{attribute 'linkalways'} 
{attribute 'no_explicit_call' := 'This FB is a CLASS and must be accessed using methods or properties'}
{attribute 'enable_dynamic_creation'}
FUNCTION_BLOCK _ETcVnColorMapSize EXTENDS EnumDatatypeBase
VAR
	localData : ETcVnColorMapSize;
	activeData : REFERENCE TO ETcVnColorMapSize;
	enumBaseDatatype : _UDINT(localData);
END_VAR

METHOD PRIVATE AddLocalEnumeration
VAR_INPUT
	Enumeration : T_MAXSTRING;
	Value : ETcVnColorMapSize;
END_VAR
AddEnumeration(Enumeration, Value);
END_METHOD

PROPERTY PUBLIC Address : PVOID
GET
Address := ADR(activeData);
END_GET
END_PROPERTY

METHOD PUBLIC ClearReference
VAR_INPUT
END_VAR
activeData REF= localData;
SetBaseDatatypeReference();
END_METHOD

METHOD PUBLIC Clone : I_Datatype
VAR
    pClone : POINTER TO _ETcVnColorMapSize;
END_VAR
pClone := __NEW(_ETcVnColorMapSize(InitialValue := Value));
Clone := pClone^;
END_METHOD

METHOD FB_init : BOOL
VAR_INPUT
	bInitRetains : BOOL; // if TRUE, the retain variables are initialized (warm start / cold start)
	bInCopyCode : BOOL;  // if TRUE, the instance afterwards gets moved into the copy code (online change)
	InitialValue : ETcVnColorMapSize;
END_VAR
localData := InitialValue;
AddBaseDatatype(enumBaseDatatype);
ClearReference();

AddLocalEnumeration('TCVN_CMS_256', ETcVnColorMapSize.TCVN_CMS_256);
AddLocalEnumeration('TCVN_CMS_65536', ETcVnColorMapSize.TCVN_CMS_65536);
END_METHOD

PROPERTY PUBLIC Identifier : T_MAXSTRING
GET
Identifier := 'ETcVnColorMapSize';
END_GET
END_PROPERTY

METHOD IsEnumeratorValueEqual : BOOL
VAR_INPUT
	Enumerator : I_KeyValueForwardEnumerator;
END_VAR
VAR
	storedValue : ETcVnColorMapSize;
END_VAR
IF NOT Enumerator.TryGet(storedValue) THEN
	RETURN;
END_IF

IsEnumeratorValueEqual := storedValue = activeData;
END_METHOD

METHOD PUBLIC MakeReferenceTo
VAR_INPUT
	ReferenceTarget : REFERENCE TO ETcVnColorMapSize;
END_VAR
activeData REF= ReferenceTarget;
SetBaseDatatypeReference();
END_METHOD

METHOD PROTECTED SetBaseDatatypeReference
VAR_INPUT
END_VAR
enumBaseDatatype.MakeReferenceTo(activeData);
END_METHOD

PROPERTY PUBLIC Size : UDINT
GET
Size := SIZEOF(activeData);
END_GET
END_PROPERTY

METHOD TryMakeReferenceTo : BOOL
VAR_INPUT
	Target : I_Datatype;
END_VAR
VAR
	targetAsEnum : I_EnumDatatype;
	pTargetData : POINTER TO ETcVnColorMapSize;
END_VAR
IF NOT Target.TryResolveAsEnumDatatype(targetAsEnum) THEN
	RETURN;
END_IF

IF targetAsEnum.Identifier <> Identifier THEN
	RETURN;
END_IF

pTargetData := Target.Address;
activeData REF= pTargetData^;
SetBaseDatatypeReference();
TryMakeReferenceTo := TRUE;
END_METHOD

PROPERTY PUBLIC Value : ETcVnColorMapSize
GET
Value := activeData;
END_GET
SET
activeData := Value;
END_SET
END_PROPERTY

END_FUNCTION_BLOCK

(* stored: Version 1.1.0.1
   POU _ETcVnColorMapSize: Id {1ef842f2-72c7-0a74-374a-5046c3d004ec}, SpecialFunc None
   Folder Constructor: Id {99d7ec45-aa66-01e3-1838-09245b097976}
   Folder Private: Id {1741206b-5689-04f5-3e9b-019bc7eb1484}
   Folder Protected: Id {5d5b4ef5-7d41-0286-0ac9-7427c5d14e26}
   Method AddLocalEnumeration: Id {eaa17899-dd27-08d9-10ae-259d589bb393}
   Property Address: Id {512a2a53-2f64-0085-378f-cc3f0621cf79}
   Get Get: Id {8d16d9e0-4c65-0c96-16f6-239ff61ac3b6}
   Method ClearReference: Id {17219168-731d-0303-0d24-16abbbae723d}
   Method Clone: Id {10406f8b-e00e-0f52-279e-548722e9496e}
   Method FB_init: Id {663b633e-f21e-0e86-01a3-70dd16deb13f}
   Property Identifier: Id {8a4fda85-5b75-0a56-39be-789cfbce3769}
   Get Get: Id {fbb60f4a-6a38-0064-0b6c-73052abddb16}
   Method IsEnumeratorValueEqual: Id {965a596e-3f5f-06e6-322b-6028457fd108}
   Method MakeReferenceTo: Id {7e9b0104-8ce8-0a45-378a-70e648144265}
   Method SetBaseDatatypeReference: Id {b6800bb2-63f5-07e1-0cdc-d0c06850d84a}
   Property Size: Id {0e2fe27f-17cc-01b9-20d4-a9a9818bc076}
   Get Get: Id {0681b4b8-11bd-0bd8-2e43-51616b2d3783}
   Method TryMakeReferenceTo: Id {a8b2cf68-b014-0f66-1846-b27c3af8ce9d}
   Property Value: Id {e3abd3b9-5e17-0672-0262-51eb22fc9605}
   Get Get: Id {b3ca3bf3-6d12-095b-1a6b-1e86711b7250}
   Set Set: Id {e491cfef-76cc-0094-0ca6-36e3b83ccd39} *)
